PROGRAM Simulation
VAR
END_VAR


SimulationViewBindings();

END_PROGRAM

(* stored: Version 1.1.0.1, ProductVersion 3.1.4024.9
   POU Simulation: Id {5d906d4b-9516-4e23-8a16-d66aa578ea01}, SpecialFunc None *)
